FUNCTION_BLOCK Service_AIMeasure (* Basic Function Block Type *)
  (* Standard: 61499-2 *)
  (* Version 0.0, 2014-5-4, wildai, nxtControl GmbH, Template *)
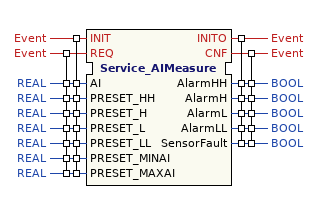
  EVENT_INPUT
    INIT WITH AI, PRESET_HH, PRESET_H, PRESET_L, PRESET_LL, PRESET_MINAI, PRESET_MAXAI; (* Initialization Request *)
    REQ WITH AI, PRESET_HH, PRESET_H, PRESET_L, PRESET_LL, PRESET_MINAI, PRESET_MAXAI; (* Normal Execution Request *)
  END_EVENT
  EVENT_OUTPUT
    INITO WITH AlarmHH, AlarmH, AlarmL, AlarmLL, SensorFault; (* Initialization Confirm *)
    CNF WITH AlarmHH, AlarmH, AlarmL, AlarmLL, SensorFault; (* Execution Confirmation *)
  END_EVENT
  VAR_INPUT
    AI : REAL;
    PRESET_HH : REAL;
    PRESET_H : REAL;
    PRESET_L : REAL;
    PRESET_LL : REAL;
    PRESET_MINAI : REAL;
    PRESET_MAXAI : REAL;
  END_VAR
  VAR_OUTPUT
    AlarmHH : BOOL;
    AlarmH : BOOL;
    AlarmL : BOOL;
    AlarmLL : BOOL;
    SensorFault : BOOL;
  END_VAR
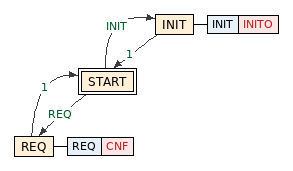
  EC_STATES
    START; (* Initial State *)
    INIT : INIT -> INITO; (* Initialization *)
    REQ : REQ -> CNF; (* Normal execution *)
  END_STATES
  EC_TRANSITIONS
    START TO INIT := INIT;
    INIT TO START := 1;
    START TO REQ := REQ;
    REQ TO START := 1;
  END_TRANSITIONS
  ALGORITHM INIT IN ST: (* Initialization algorithm *)
;

SensorFault := FALSE;
AlarmHH := FALSE;
AlarmH := FALSE;
AlarmL := FALSE;
AlarmLL := FALSE;
  END_ALGORITHM
  ALGORITHM REQ IN ST: (* Normally executed algorithm *)
;
IF AI < PRESET_MINAI OR AI > PRESET_MAXAI THEN
	SensorFault := TRUE;
	AlarmHH := FALSE;
	AlarmH := FALSE;
	AlarmL := FALSE;
	AlarmLL := FALSE;
ELSE
	SensorFault := FALSE;
	IF AI >= PRESET_HH THEN
		AlarmHH := TRUE;
		AlarmH := FALSE;
		AlarmL := FALSE;
		AlarmLL := FALSE;
	ELSIF AI < PRESET_H AND AI >= PRESET_H THEN
		AlarmHH := FALSE;
		AlarmH := TRUE;
		AlarmL := FALSE;
		AlarmLL := FALSE;
	ELSIF AI <= PRESET_L AND AI > PRESET_LL THEN
		AlarmHH := FALSE;
		AlarmH := FALSE;
		AlarmL := TRUE;
		AlarmLL := FALSE;
	ELSIF AI <= PRESET_LL THEN
		AlarmHH := FALSE;
		AlarmH := FALSE;
		AlarmL := FALSE;
		AlarmLL := TRUE;
	ELSE
		AlarmHH := FALSE;
		AlarmH := FALSE;
		AlarmL := FALSE;
		AlarmLL := FALSE;
	END_IF;
END_IF;
  END_ALGORITHM
END_FUNCTION_BLOCK
